// TIA Portal V19 export
TYPE "SpeedMotor_Sts"
// stored: Access Published
   STRUCT
      AlarmPresence : Bool;   // Cumulative alarm presence
      WarningPresence : Bool;   // Cumulative warning presence
      Enabled : Bool;   // Axis enabled
      Standstill : Bool;   // Axis standstill
      AtProgrammedSpeed : Bool;   // Axis at programmed speed
      MoveMinusPermitted : Bool;   // Move minus permitted
      MovePlusPermitted : Bool;   // Move plus permitted
      ActualVelocity : LReal;   // Aactual velocity (rpm)
   END_STRUCT;
END_TYPE
